INTERFACE I_FallibleDword


PROPERTY Error : BOOL
GET
END_GET
END_PROPERTY


PROPERTY Value : DWORD
GET
END_GET
END_PROPERTY

END_INTERFACE

(* stored: Version 1.1.0.1
   Itf I_FallibleDword: Id {a1b2c3d4-0002-4001-8001-000000000011}
   Property Error: Id {a1b2c3d4-0002-4001-8001-000000000012}
   Get Get: Id {a1b2c3d4-0002-4001-8001-000000000013}
   Property Value: Id {a1b2c3d4-0002-4001-8001-000000000014}
   Get Get: Id {a1b2c3d4-0002-4001-8001-000000000015} *)
